// TIA Portal V19 export
FUNCTION "FC_FW_SCHIEBEN" : Void   // FC21, STL
{ S7_Optimized_Access := 'FALSE' }
AUTHOR : MS
// stored: AutoNumber false
   VAR_TEMP
      count_FW : Byte;
      FW_DB_1 : Word;
      FW_DB_2 : Word;
      QT_DB : Word;
      CHK_POS_min : Int;
      CHK_POS_max : Int;
      CHK_Z_min : DInt;
      CHK_Z_max : DInt;
      CHK_POS : Int;
      CHK_Z : Int;
      PosFW : DInt;
      SchiebePos : DInt;
      SchiePos : Byte;
      schieben : Bool;
      count : Int;
      Rcount : Byte;   // Reihenzähler QT
      ZielBereich : DInt;
      Schwerpunkt : Byte;
      ziel : Int;
      FW_Nr : Int;
      erlaubt : Bool;
      Offset : Bool;
   END_VAR
BEGIN

NETWORK
TITLE = 
      L     "DB_ANLAGE".config.ANZ_FW;
      L     1;
      -I;
      T     #count_FW;
ret:  L     #count_FW;
      L     0;
      <=I;
      JC    NW3;

      L     #count_FW;
      L     10;
      +I;
      T     #FW_DB_1;
      L     1;
      +I;
      T     #FW_DB_2;

//------------------------
//SCHIEBEMERKER RESET
//------------------------
      OPN   DB [#FW_DB_1];
      L     %DBW30;  //Liegt Befehl an ?
      L     0;
      ==I;
      A     %DBX13.0;  //"DI_FW_1".ZST.schieben
      R     %DBX13.0;  //"DI_FW_1".ZST.schieben

      OPN   DB [#FW_DB_2];
      L     %DBW30;  //Liegt Befehl an ?
      L     0;
      ==I;
      A     %DBX13.0;  //"DI_FW_2".ZST.schieben
      R     %DBX13.0;  //"DI_FW_2".ZST.schieben

//------------------------
//FW rückwärts schieben
//------------------------
      OPN   DB [#FW_DB_1];

      AN    %DBX1.6;  //"DBI_FW_1".ZST.Auto
      AN    %DBX1.5;  //"DBI_FW_1".ZST.Auto_Stop
      AN(;
      A     %DBX1.4;  //"DI_FW_1".ZST.Hand
      A     %DBX13.5;  //"DI_FW_1".ZST.schieben_erlaubt
      );
      ON    %DBX0.0;  //"DBI_FW_1".ZST.BEREIT
      O     %DBX0.1;  //aktiv
      O     %DBX0.2;  //Fehler
      O     %DBX13.0;  //"DI_FW_1".ZST.schieben
      JC    NW2;

      OPN   DB [#FW_DB_2];  //keine bzw. andere Fahrtrichtung
      L     0;
      L     %DBB351;  //"DI_FW_2".TMP.ZielPos
      ==I;
      ON    %DBX0.7;  //"DBI_FW_2".ZST.RUECKWAERTS_AKT
      JC    NW2;

      L     %DBB351;  //"DI_FW_2".TMP.ZielPos
      L     "DB_POS".LENG;
      *I;
      L     "DB_POS".Offset;
      +I;
      SLD   3;
      LAR1;
      OPN   "DB_POS";
      L     DBD [AR1, P#22.0];  //Position des Zielbades in Inkrementen
      OPN   DB [#FW_DB_1];
      L     %DBD198;  //"DI_FW_1".PAR.Fahrt.Abstand_vor
      -D;
//      L     DBW  234                    //"DI_FW_1".PAR.Fahrt.SoftOffset
//      -D
      OPN   DB [#FW_DB_2];
      L     %DBD212;  //"DI_FW_2".PAR.Fahrt.Bereich_Pos
      -D;
      T     #SchiebePos;
      OPN   DB [#FW_DB_1];
      L     %DBD4;  //"DI_FW_1".ZST.PosInc
      >=D;
      JC    NW2;
      OPN   DB [#FW_DB_1];
      L     #SchiebePos;
      L     %DBD212;  //"DI_FW_1".PAR.Fahrt.Bereich_Pos
      -D;
      T     #SchiebePos;

      L     0;
      L     %DBW396;  //"DI_FW_1".TMP.nexQuelle
      ==I;
      JC    noRe;
      L     "DB_POS".LENG;
      *I;
      L     "DB_POS".Offset;
      +I;
      SLD   3;
      LAR1;
      OPN   "DB_POS";
      L     #SchiebePos;
      L     DBD [AR1, P#22.0];  //Position des Zielbades in Inkrementen
      >=D;
      JC    NW2;

noRe: OPN   DB [#FW_DB_1];
      L     %DBB2;  //"DBI_FW_1".ZST.POSITION
retR: T     #count;
      OPN   DB [#FW_DB_1];
      L     %DBB194;  //"DI_FW_1".PAR.Fahrt.FAHRBEREICH_MIN
      <I;
      JC    NW2;

      L     #count;
      L     "DB_POS".LENG;
      *I;
      L     "DB_POS".Offset;
      +I;
      SLD   3;
      LAR1;
      OPN   "DB_POS";
      L     #SchiebePos;
      L     DBD [AR1, P#22.0];  //BadPosition
      >=D;
      JC    TakR;

      L     #count;
      L     1;
      -I;
      JU    retR;

TakR: OPN   DB [#FW_DB_1];
      S     %DBX13.0;  //"DI_FW_1".ZST.schieben
      L     16#FF01;
      T     %DBW30;  //Befehlskennung
      L     #count;
      T     %DBB32;  //FW Ziel
      L     #SchiebePos;
      T     %DBD38;  //"DI_FW_1".ZST.SchiebeInc


NETWORK
TITLE = 
//------------------------
//FW vorwärts schieben
//------------------------
NW2:  OPN   DB [#FW_DB_2];
      AN    %DBX1.6;  //"DBI_FW_2".ZST.Auto
      AN    %DBX1.5;  //"DBI_FW_2".ZST.Auto_Stop
      AN    %DBX1.4;  //"DI_FW_2".ZST.Hand
      ON    %DBX13.5;  //"DI_FW_2".ZST.schieben_erlaubt
      ON    %DBX0.0;  //"DBI_FW_2".ZST.BEREIT
      O     %DBX0.1;  //aktiv
      O     %DBX0.2;  //Fehler
      O     %DBX13.0;  //"DI_FW_2".ZST.schieben
      JC    nxt;

      OPN   DB [#FW_DB_1];
      L     0;
      L     %DBB351;  //"DI_FW_1".TMP.ZielPos
      ==I;
      ON    %DBX0.6;  //"DBI_FW_1".ZST.VORWAERTS_AKT
      JC    nxt;

      L     %DBB351;  //"DI_FW_1".TMP.ZielPos
      L     "DB_POS".LENG;
      *I;
      L     "DB_POS".Offset;
      +I;
      SLD   3;
      LAR1;
      OPN   "DB_POS";
      L     DBD [AR1, P#22.0];  //Position des Zielbades in Inkrementen
      OPN   DB [#FW_DB_1];
      L     %DBD198;  //"DI_FW_1".PAR.Fahrt.Abstand_vor
      +D;
//      L     DBW  234                    //"DI_FW_1".PAR.Fahrt.SoftOffset
//      +D
      OPN   DB [#FW_DB_2];
      L     %DBD212;  //"DI_FW_2".PAR.Fahrt.Bereich_Pos
      +D;
      T     #SchiebePos;
      L     %DBD4;  //"DI_FW_2".ZST.PosInc
      <=D;
      JC    nxt;
      OPN   DB [#FW_DB_1];
      L     #SchiebePos;
      L     %DBD212;  //"DI_FW_1".PAR.Fahrt.Bereich_Pos
      +D;
      T     #SchiebePos;

      OPN   DB [#FW_DB_2];
      L     0;
      L     %DBW396;  //"DI_FW_1".TMP.nexQuelle
      ==I;
      JC    noLi;
      L     "DB_POS".LENG;
      *I;
      L     "DB_POS".Offset;
      +I;
      SLD   3;
      LAR1;
      OPN   "DB_POS";
      L     #SchiebePos;
      L     DBD [AR1, P#22.0];  //Position des Zielbades in Inkrementen
      <=D;
      JC    nxt;

noLi: OPN   DB [#FW_DB_2];
      L     %DBB2;  //"DBI_FW_2".ZST.POSITION
retV: T     #count;
      OPN   DB [#FW_DB_2];
      L     %DBB195;  //"DI_FW_2".PAR.Fahrt.FAHRBEREICH_MAX
      >I;
      JC    nxt;

      L     #count;
      L     "DB_POS".LENG;
      *I;
      L     "DB_POS".Offset;
      +I;
      SLD   3;
      LAR1;
      OPN   "DB_POS";
      L     #SchiebePos;
      L     DBD [AR1, P#22.0];  //BadPosition
      <=D;
      JC    TakL;

      L     #count;
      L     1;
      +I;
      JU    retV;

TakL: OPN   DB [#FW_DB_2];
      S     %DBX13.0;  //"DI_FW_2".ZST.schieben
      L     16#FF01;
      T     %DBW30;  //Befehlskennung
      L     #count;
      T     %DBB32;  //FW Ziel
      L     #SchiebePos;
      T     %DBD38;  //"DI_FW_1".ZST.SchiebeInc

nxt:  L     #count_FW;
      DEC   1;
      T     #count_FW;
      JU    ret;


NETWORK
TITLE = QT schiebt FW
NW3:  NOP   0;

      L     0;
      T     #SchiebePos;

//Es gibt keine QT
      L     0;
      L     "DB_ANLAGE".config.ANZ_QT;
      >=I;
      BEC;

//QT Prüfschleife

      L     30;
      +I;
reQ:  T     #QT_DB;

      OPN   DB [#QT_DB];
      L     %DBB104;  //"DBI_QT_1".TMP.ZIEL_REIHE QT will nicht fahren
      L     0;
      ==I;
      O(;
      L     %DBB100;  //"DI_QT_1".TMP.ZIEL_POS
      L     0;
      ==I;
      );
      JC    nxtQ;

//Ermittlung gesperrter Bereich um QT-Zielposition
      OPN   DB [#QT_DB];
      L     0;
      T     #Rcount;

reR:  L     #Rcount;
      L     5;
      >=I;
      JC    nxtQ;

      OPN   DB [#QT_DB];
      L     #Rcount;
      L     60;
      +D;
      SLD   3;
      LAR1;

      L     0;
      L     DBB [AR1, P#0.0];  //"DBI_QT_1".PAR.POS1..5
      ==I;
      JC    nxtQ;
      T     #CHK_POS;

      L     "DB_POS".LENG;
      *I;
      L     "DB_POS".Offset;
      +I;
      SLD   3;
      LAR1;
      OPN   "DB_POS";
      L     DBD [AR1, P#22.0];  //BadPosition
      L     DBW [AR1, P#26.0];  //Abstand_vor
      +D;
      T     #CHK_Z_max;

      L     DBD [AR1, P#22.0];  //BadPosition
      L     DBW [AR1, P#28.0];  //Abstand_rck
      -D;
      T     #CHK_Z_min;

      L     DBB [AR1, P#3.0];  //Schiebepos
      T     #SchiePos;

      L     "DB_ANLAGE".config.ANZ_FW;
      L     10;
      +I;
reF:  T     #FW_DB_1;

      OPN   DB [#FW_DB_1];
      AN    %DBX1.6;  //"DBI_FW_1".ZST.Auto
      AN    %DBX1.5;  //"DBI_FW_1".ZST.Auto_Stop
//  UN    DBX    1.4                  //"DI_FW_2".ZST.Hand
      ON    %DBX13.5;  //"DI_FW_2".ZST.schieben_erlaubt
      ON    %DBX0.0;  //"DBI_FW_1".ZST.BEREIT
      O     %DBX0.1;  //aktiv
      O     %DBX0.2;  //Fehler
      O     %DBX13.0;  //"DI_FW_1".ZST.schieben
      JC    nxtF;
      R     #schieben;

      OPN   DB [#FW_DB_1];
      L     %DBD4;  //"DI_FW_1".ZST.PosInc
      T     #PosFW;
      L     %DBD220;  //"DI_FW_1".PAR.Fahrt.Bereich_Ziel
      T     #ZielBereich;

//      L     #CHK_Z_max
//      L     #ZielBereich
//      +D
//      T     #CHK_Z_max

      L     #PosFW;
      L     #CHK_Z_max;
      >=D;
      JC    nxtF;

//      L     #CHK_Z_min
//      L     #ZielBereich
//      -D
//      T     #CHK_Z_min

      L     #PosFW;
      L     #CHK_Z_min;
      <=D;
      JC    nxtF;
      S     #schieben;

      AN    #schieben;
      JC    nxtF;

      L     #CHK_Z_max;
      L     #ZielBereich;
      +D;
      T     #CHK_Z_max;

      L     #CHK_Z_min;
      L     #ZielBereich;
      -D;
      T     #CHK_Z_min;

      L     0;
      L     #SchiePos;  //keine Schiebepos definiert
      ==I;  //deshalb in Richtung Schwerpunkt schieben
      =     #Offset;
      JC    such;

fnd:  L     #SchiePos;
      T     #ziel;
      L     0;
      ==I;
      JC    nxtF;

      OPN   DB [#FW_DB_1];
      L     0;
      L     %DBW396;  //"DI_FW_1".TMP.nexQuelle
      ==I;
      JC    noQ;
      L     "DB_POS".LENG;
      *I;
      L     "DB_POS".Offset;
      +I;
      SLD   3;
      LAR1;
      OPN   "DB_POS";
      L     #CHK_Z_min;
      L     DBD [AR1, P#22.0];  //Position des Zielbades in Inkrementen
      <=D;
      O(;
      L     #CHK_Z_max;
      L     DBD [AR1, P#22.0];  //Position des Zielbades in Inkrementen
      >=D;
      );
      JC    nxtF;

noQ:  L     #FW_DB_1;
      +     -10;
      T     #FW_Nr;

      CALL  "FC_FW_Befehl_ok"
      ( FW_Nr    := #FW_Nr,
        kl_Z     := #ziel,
        Gr_Z     := #ziel,
        QT_Check := FALSE,
        Ablassen := FALSE,
        vor      := FALSE,
        chk_on   := FALSE,
        erlaubt  := #erlaubt
      );

      AN    #erlaubt;
      JC    nxtF;

      OPN   DB [#FW_DB_1];
      L     16#F001;
      AN    #Offset;
      JC    toPo;
      L     16#FF01;
toPo: T     %DBW30;  //Befehlskennung
      L     #SchiePos;
      T     %DBB32;  //FW Ziel
      L     #SchiebePos;
      T     %DBD38;  //"DI_FW_1".ZST.SchiebeInc

nxtF: L     #FW_DB_1;
      L     11;
      <=I;
      JC    nxR;

      L     #FW_DB_1;
      L     1;
      -I;
      T     #FW_DB_1;
      JU    reF;

nxtQ: L     #QT_DB;
      L     31;
      <=I;
      BEC;

      L     #QT_DB;
      L     1;
      -I;
      JU    reQ;

nxR:  L     #Rcount;
      L     1;
      +I;
      T     #Rcount;
      JU    reR;

//Suche nach Schiebepos in Richtung Schwerpunkt
such: L     #CHK_POS;
      T     #SchiePos;

      OPN   DB [#FW_DB_1];
      L     0;
      L     %DBW396;  //"DI_FW_1".TMP.nexQuelle
      ==I;
      JC    spnt;
      JU    pkt;

spnt: OPN   DB [#FW_DB_1];
      L     %DBB194;  //"DI_FW_1".PAR.Fahrt.FAHRBEREICH_MIN
      L     %DBB195;  //"DI_FW_1".PAR.Fahrt.FAHRBEREICH_MAX
      +I;
      L     2;
      /I;
pkt:  T     #Schwerpunkt;

      L     #CHK_POS;
      L     #Schwerpunkt;
      >=I;
      JC    Srck;  //Schiebe rückwärts

Svor: L     #SchiePos;
      L     1;
      +I;
      T     #SchiePos;

      L     "DB_POS".LENG;
      *I;
      L     "DB_POS".Offset;
      +I;
      SLD   3;
      LAR1;
      OPN   "DB_POS";
      L     DBD [AR1, P#22.0];  //BadPosition
      L     #CHK_Z_max;
      <D;
      JC    Svor;
      T     #SchiebePos;
      JU    fnd;

Srck: L     #SchiePos;
      L     1;
      -I;
      T     #SchiePos;

      L     "DB_POS".LENG;
      *I;
      L     "DB_POS".Offset;
      +I;
      SLD   3;
      LAR1;
      OPN   "DB_POS";
      L     DBD [AR1, P#22.0];  //BadPosition
      L     #CHK_Z_min;
      >D;
      JC    Srck;
      T     #SchiebePos;
      JU    fnd;

END_FUNCTION
